Staubli VAL3: Exam_2025_59333.pjx

--- Exam_2025_59333.pjx ---
Parameters version=s7.11.2 stackSize=5000 millimeterUnit=true
Program file=Empilement.pgx
Program file=Exam_Robot.pgx
Program file=Initialisation.pgx
Program file=Pause.pgx
Program file=Prise.pgx
Program file=start.pgx
Program file=stop.pgx
Data file=Exam_2025_59333.dtx

--- Exam_2025_59333.dtx ---
mdesc mNomSpeed
mdesc mRapide = {accel=75, vel=75, decel=75}
mdesc mLent = {accel=10, vel=10, decel=10}
pointRx pP1 = {fatherId=world[0]}
jointRx jDepart
num nDistancePiece = 80
num nDistanceLigne = 160
num nPieceLigne = 3
num nLigne
bool bDCY = true
num nHauteurPiece = 100
tool tPince = {z=100, fatherId=flange[0], ioLink=valve1}
trsf trAppro = {z=-100}
trsf trDecalPiece
trsf trDecalHauteur
num nCycles
num nDebut
num nFin

--- Pause.pgx ---
program Pause(point x_pPoint (dimensions=1))
begin
  movej(appro(x_pPoint,trAppro),tPince,mRapide)
  movel(x_pPoint,tPince,mLent)
  open(tPince)
  movel(appro(x_pPoint,trAppro),tPince,mRapide)
  close(tPince)

end

--- Prise.pgx ---
program Prise(point x_pPoint (dimensions=1))
begin
  movej(appro(x_pPoint,trAppro),tPince,mRapide)
  open(tPince)
  movel(x_pPoint,tPince,mLent)
  close(tPince)
  movel(appro(x_pPoint,trAppro),tPince,mLent)
end
